FUNCTION_BLOCK ModbusReadBits EXTENDS ModbusIo
VAR_INPUT
END_VAR
VAR_OUTPUT
	b0: BOOL;
	b1: BOOL;
	b2: BOOL;
	b3: BOOL;
	b4: BOOL;
	b5: BOOL;
	b6: BOOL;
	b7: BOOL;
	b8: BOOL;
	b9: BOOL;
	b10: BOOL;
	b11: BOOL;
	b12: BOOL;
	b13: BOOL;
	b14: BOOL;
	b15: BOOL;
END_VAR
VAR
END_VAR

SUPER^();

PROPERTY ValueWord : WORD
GET
ValueWord := 0;
IF b0 THEN
	ValueWord := ValueWord OR 16#0001;
END_IF
IF b1 THEN
	ValueWord := ValueWord OR 16#0002;
END_IF
IF b2 THEN
	ValueWord := ValueWord OR 16#0004;
END_IF
IF b3 THEN
	ValueWord := ValueWord OR 16#0008;
END_IF
IF b4 THEN
	ValueWord := ValueWord OR 16#0010;
END_IF
IF b5 THEN
	ValueWord := ValueWord OR 16#0020;
END_IF
IF b6 THEN
	ValueWord := ValueWord OR 16#0040;
END_IF
IF b7 THEN
	ValueWord := ValueWord OR 16#0080;
END_IF
IF b8 THEN
	ValueWord := ValueWord OR 16#0100;
END_IF
IF b9 THEN
	ValueWord := ValueWord OR 16#0200;
END_IF
IF b10 THEN
	ValueWord := ValueWord OR 16#0400;
END_IF
IF b11 THEN
	ValueWord := ValueWord OR 16#0800;
END_IF
IF b12 THEN
	ValueWord := ValueWord OR 16#1000;
END_IF
IF b13 THEN
	ValueWord := ValueWord OR 16#2000;
END_IF
IF b14 THEN
	ValueWord := ValueWord OR 16#4000;
END_IF
IF b15 THEN
	ValueWord := ValueWord OR 16#8000;
END_IF
END_GET
SET
b0 := (ValueWord AND 16#0001) <> 0;
b1 := (ValueWord AND 16#0002) <> 0;
b2 := (ValueWord AND 16#0004) <> 0;
b3 := (ValueWord AND 16#0008) <> 0;
b4 := (ValueWord AND 16#0010) <> 0;
b5 := (ValueWord AND 16#0020) <> 0;
b6 := (ValueWord AND 16#0040) <> 0;
b7 := (ValueWord AND 16#0080) <> 0;
b8 := (ValueWord AND 16#0100) <> 0;
b9 := (ValueWord AND 16#0200) <> 0;
b10 := (ValueWord AND 16#0400) <> 0;
b11 := (ValueWord AND 16#0800) <> 0;
b12 := (ValueWord AND 16#1000) <> 0;
b13 := (ValueWord AND 16#2000) <> 0;
b14 := (ValueWord AND 16#4000) <> 0;
b15 := (ValueWord AND 16#8000) <> 0;
END_SET
END_PROPERTY

END_FUNCTION_BLOCK

(* stored: Version 1.1.0.1, ProductVersion 3.1.4024.6
   POU ModbusReadBits: Id {5e7aab4f-4075-4a76-b76a-9822912767b6}, SpecialFunc None
   Property ValueWord: Id {bcc57c69-d637-4c03-8361-57d5c423fdc3}
   Get Get: Id {c6873f3c-2f53-4f68-8b6f-9029b0403e14}
   Set Set: Id {3ae1f94e-cd7d-4b1c-ab15-bf10b658fe0a} *)
